TYPE ST_Cylinder :
STRUCT
END_STRUCT
END_TYPE

(* stored: Version 1.1.0.1, ProductVersion 3.1.4024.12
   DUT ST_Cylinder: Id {777eee00-50aa-4df4-949a-13c0c9701e74} *)
